FUNCTION_BLOCK fbHMIBit
VAR_INPUT
	bInToggle:BOOL;
	bInLatch:BOOL;
END_VAR
VAR_OUTPUT
END_VAR
VAR
	RTrigHMI:R_TRIG;
END_VAR
VAR_IN_OUT
	bHMI:BOOL;
	bPLC:BOOL;
END_VAR

RTrigHMI(CLK:=bHMI , Q=> );

IF bIntoggle THEN
	IF RTrigHMI.Q AND NOT bPLC THEN
		bPLC:=1;
	END_IF
	
	IF   RTrigHMI.Q AND bPLC THEN
		bPLC:=0;
	END_IF
ELSE
	bPLC:=bHMI;
END_IF

END_FUNCTION_BLOCK

(* stored: Version 1.1.0.1, ProductVersion 3.1.4024.11
   POU fbHMIBit: Id {54195508-1a4e-45f3-8be6-b212bf29d5eb}, SpecialFunc None *)
